Omron CX-Programmer project NewProject (CX-Programmer 9.73)

# PLC AutoRCG: CP1L M

## Global symbols (name address type ; comment)
0.01 BOOL  ; ENTRY-SENSOR
100.05 BOOL  ; SIGNAL-LIGHT_2
100.00 BOOL  ; GATE-MOTOR_CLOSE
100.04 BOOL  ; SIGNAL-LIGHT_1
100.02 BOOL  ; BUZZER_1
0.00 BOOL  ; ON START
0.02 BOOL  ; EXIT-SENSOR
0.03 BOOL  ; EMERGENCY-BUTTON
100.01 BOOL  ; GATE-MOTOR_OPEN
100.03 BOOL  ; BUZZER_2
T0001 BOOL  ; TIMER_1
T0002 BOOL  ; TIMER_2
W100.00 BOOL  ; 0
W100.01 BOOL  ; 1
W100.02 BOOL  ; 2
W100.03 BOOL  ; EMERGENCY

## Program NewProgram1 (cyclic task 0)

### Section Section1

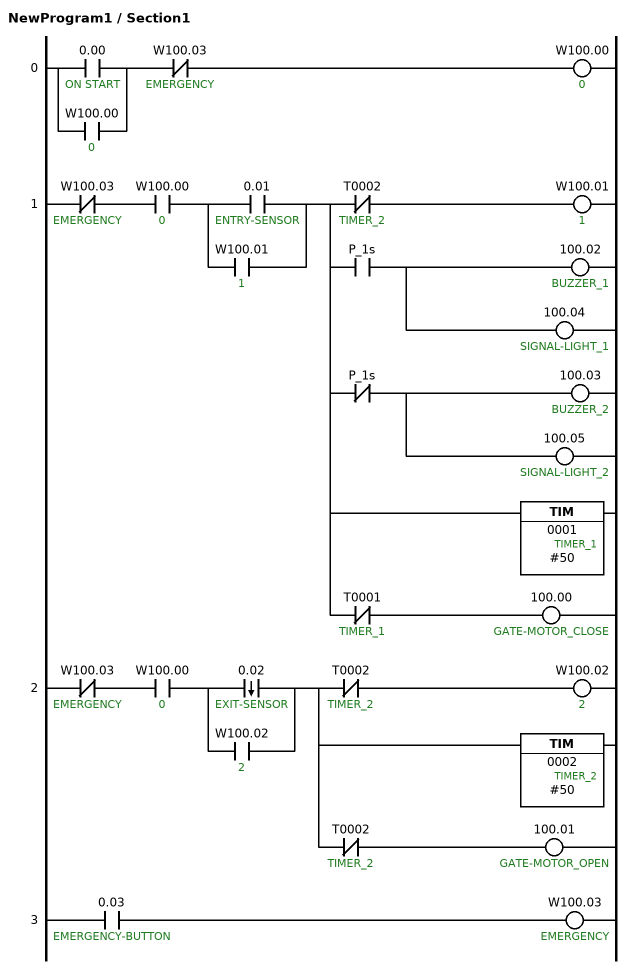
; rung 0
LD 0.00  ; ON START
OR W100.00  ; 0
ANDNOT W100.03  ; EMERGENCY
OUT W100.00  ; 0
; rung 1
LDNOT W100.03  ; EMERGENCY
AND W100.00  ; 0
LD 0.01  ; ENTRY-SENSOR
OR W100.01  ; 1
ANDLD
OUT TR0
ANDNOT T0002  ; TIMER_2
OUT W100.01  ; 1
LD TR0
AND P_1s
OUT 100.02  ; BUZZER_1
OUT 100.04  ; SIGNAL-LIGHT_1
LD TR0
ANDNOT P_1s
OUT 100.03  ; BUZZER_2
OUT 100.05  ; SIGNAL-LIGHT_2
LD TR0
TIM 0001 #50  ; TIMER_1
ANDNOT T0001  ; TIMER_1
OUT 100.00  ; GATE-MOTOR_CLOSE
; rung 2
LDNOT W100.03  ; EMERGENCY
AND W100.00  ; 0
%LD 0.02  ; EXIT-SENSOR
OR W100.02  ; 2
ANDLD
OUT TR0
ANDNOT T0002  ; TIMER_2
OUT W100.02  ; 2
LD TR0
TIM 0002 #50  ; TIMER_2
ANDNOT T0002  ; TIMER_2
OUT 100.01  ; GATE-MOTOR_OPEN
; rung 3
LD 0.03  ; EMERGENCY-BUTTON
OUT W100.03  ; EMERGENCY

### Section END
; rung 0
END(001)